SUBAPPLICATION RedGreenBackground4C (* Hintergrundfarbe (TRUE -> Rot, FALSE -> Grün) für 4 Objekte (Kompakt) *)
  (* Standard: 61499-2 *)
  (* Version 1.0, 2022-11-10, franz, Meisterschulen am Ostbahnhof *)
  PACKAGE MyLib::sys;
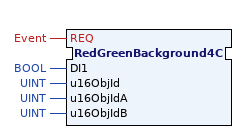
  EVENT_INPUT
    REQ; (* Normal Execution Request *)
  END_EVENT
  VAR_INPUT
    DI1 : BOOL; (* Selector *)
    u16ObjId : UINT; (* Object ID Softkey *)
    u16ObjIdA : UINT; (* Object ID AUX *)
    u16ObjIdB : UINT;
  END_VAR
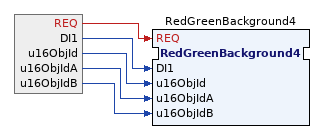
  SUBAPPS
    RedGreenBackground4 : MyLib::sys::RedGreenBackground4;
  END_SUBAPPS
  EVENT_CONNECTIONS
    REQ TO RedGreenBackground4.REQ;
  END_CONNECTIONS
  DATA_CONNECTIONS
    DI1 TO RedGreenBackground4.DI1;
    u16ObjId TO RedGreenBackground4.u16ObjId;
    u16ObjIdA TO RedGreenBackground4.u16ObjIdA;
    u16ObjIdB TO RedGreenBackground4.u16ObjIdB;
  END_CONNECTIONS
END_SUBAPPLICATION
